ABB RobotStudio station: TP3_20201209-173036.rsstn

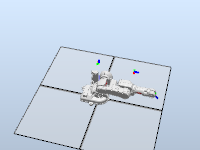
Station TP3 (saved by RobotStudio 20.2.9116.0)
Controller IRB_140_6kg_0.81m
  mechanical unit ROB_1: IRB140_6_81_C_03, 6 joints, base frame (0, 0, 0) mm
Layout (positions relative to the parent item):
  - IRB140_6_81_C_03 [mechanism, from Robots\IRB140_6_81_C_G_03.rslib] at (0, 0, 0) mm; joint values [0, 1.5705, -1.5702, 0, 0.7851, 0] (rad or m)
Targets, tools, work objects and paths stored in the station, written as RAPID:
! task T_ROB1
MODULE Module1
  CONST robtarget PosiconSingularidadCodo:=[[855.961941244,0,306.038043953],[0.382683437,0.000000096,0.923879531,0.00000004],[-1,0,0,0],[9E+09,9E+09,9E+09,9E+09,9E+09,9E+09]];
  CONST robtarget PosicionSingularidadBrazo:=[[0.000036644,0.00000422,746.110027233],[0.382683497,0.000000022,0.000000044,0.923879506],[0,-3,-1,0],[9E+09,9E+09,9E+09,9E+09,9E+09,9E+09]];
  CONST robtarget PosicionSingularidadMunieca:=[[515,0,712],[0.707106781,0.000000042,0.707106781,0.000000042],[0,0,0,0],[9E+09,9E+09,9E+09,9E+09,9E+09,9E+09]];
  PROC main()
  ENDPROC
ENDMODULE

